Fanuc KAREL source: READ_DICT_V.kl

PROGRAM T
%NOLOCKGROUP
VAR
 v0 : STRING[40]
 v1 : INTEGER
 v2 : ARRAY[10] OF STRING[40]
 v3 : ARRAY[10] OF STRING[40]
 v4 : INTEGER
BEGIN
 READ_DICT_V(v0, v1, v2, v3, v4)
END T
